// TIA Portal V20 export
TYPE "typeEmHomedCheck"
// stored: Access Published, Namespace Unit1.Em2
   STRUCT
      cmElectrodeFixRightUnit : Bool;
      cmElectrodeFixLeftUnit : Bool;
      cmUwSemiSplicerVacuumUnit : Bool;
      cmElectrodeCutterFwdBwd : Bool;
      cmSplicingModuleMoverUnit : Bool;
      cmElectrodeHolderMoverUnit : Bool;
      cmTapeUnit : Bool;
      cmStopperFwdBwd : Bool;
      cmSupportUnit : Bool;
   END_STRUCT;
END_TYPE
